Universal Robots PolyScope program: presa_e_rilascio.urp

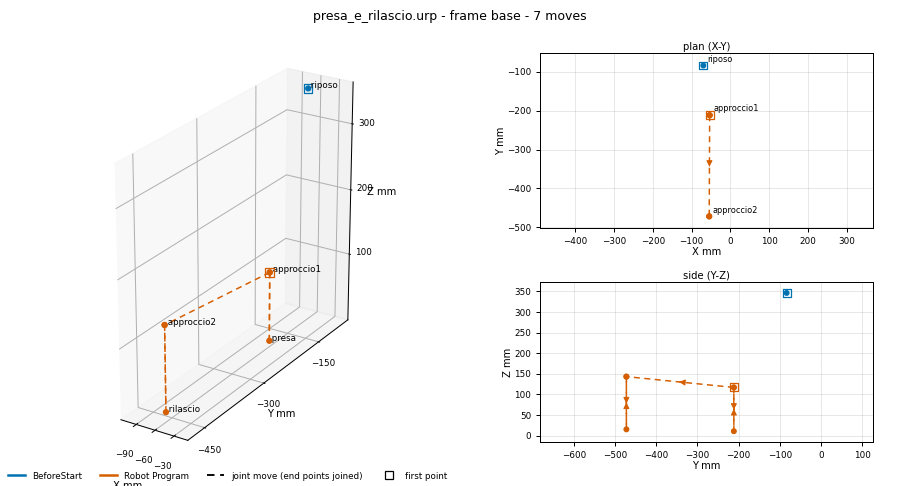
[picture p0: tool path of presa_e_rilascio.urp in frame base, 7 of 7 moves have a stored position in this frame; points joined in program order, loops and branches not executed]
Program presa_e_rilascio (installation=default directory=/programs createdIn=3.15.8.106339 lastSavedIn=3.15.8.106339 robotSerialNumber=2021330429)
Calibrated DH parameters: a=[-0.000156, -0.236402, -0.171625, 0.000006, -0.000047, 0]; d=[0.151683, 29.702709, 78.973085, -108.563557, 0.085229, 0.082167]; alpha=[1.57015, 0.001987, 0.001164, 1.571718, -1.571778, 0]; deltaTheta=[-0.000066, 0.24449, 0.39032, -0.635025, 0.000068, -0.000043]
BeforeStart
  MoveJ speed 60 deg/s, acceleration 80 deg/s^2 (useActiveTCP=true)
    Waypoint riposo: TCP in base x=-69.7 y=-83.46 z=346.387 mm, rx=-0.1858 ry=2.903 rz=-0.614 rad; joints [277.762, -45.293, -63.599, -136.482, 97.736, 362.044] deg; flange x=-99.442 y=-22.232 z=487.863 mm, rx=-0.1858 ry=2.903 rz=-0.614 rad
Robot Program (runOnlyOnce=false)
  MoveJ speed 60 deg/s, acceleration 80 deg/s^2 (useActiveTCP=true)
    Waypoint approccio1: TCP in base x=-53.385 y=-211.554 z=117.085 mm, rx=-0.0713 ry=3.1104 rz=0.0249 rad; joints [284.51, -64.741, -119.374, -86.315, 91.916, 371.806] deg; flange x=-58.082 y=-214.172 z=273.993 mm, rx=-0.0713 ry=3.1104 rz=0.0249 rad
    Waypoint presa: TCP in base x=-53.406 y=-211.507 z=10.879 mm, rx=-0.0712 ry=3.1103 rz=0.0251 rad; joints [284.47, -77.457, -143.252, -49.727, 91.95, 371.797] deg; flange x=-58.107 y=-214.145 z=167.786 mm, rx=-0.0712 ry=3.1103 rz=0.0251 rad
    URCap Gripper Activate (Robotiq_Grippers, Robotiq Inc.) dataModel(ResetAndActivateKey=false)
    URCap Gripper (Robotiq_Grippers, Robotiq Inc.) dataModel(position=100.0, force=100.0, speed=100.0, positionInDouble=100.0, forceInDouble=100.0, speedInDouble=100.0, slaveIds=[9], blocking=true)
    Waypoint approccio1: TCP in base x=-53.385 y=-211.554 z=117.085 mm, rx=-0.0713 ry=3.1104 rz=0.0249 rad; joints [284.51, -64.741, -119.374, -86.315, 91.916, 371.806] deg; flange x=-58.082 y=-214.172 z=273.993 mm, rx=-0.0713 ry=3.1104 rz=0.0249 rad
    Waypoint approccio2: TCP in base x=-54.566 y=-472.294 z=143.32 mm, rx=0.1164 ry=3.1211 rz=-0.0254 rad; joints [276.657, -133.101, -33.078, -102.673, 91.021, 370.841] deg; flange x=-57.324 y=-469.636 z=300.273 mm, rx=0.1164 ry=3.1211 rz=-0.0254 rad
    Waypoint rilascio: TCP in base x=-54.524 y=-472.289 z=15.377 mm, rx=0.1163 ry=3.1211 rz=-0.0253 rad; joints [276.679, -135.071, -64.449, -69.336, 91.045, 370.896] deg; flange x=-57.282 y=-469.647 z=172.331 mm, rx=0.1163 ry=3.1211 rz=-0.0253 rad
    URCap Gripper (Robotiq_Grippers, Robotiq Inc.) dataModel(position=0.0, force=100.0, speed=100.0, positionInDouble=0.0, forceInDouble=100.0, speedInDouble=100.0, slaveIds=[9], blocking=true)
    Waypoint approccio2: TCP in base x=-54.566 y=-472.294 z=143.32 mm, rx=0.1164 ry=3.1211 rz=-0.0254 rad; joints [276.657, -133.101, -33.078, -102.673, 91.021, 370.841] deg; flange x=-57.324 y=-469.636 z=300.273 mm, rx=0.1164 ry=3.1211 rz=-0.0254 rad
